(* CoDeSys 2.3.9.62 project: udptest.pro *)
(* Libraries: SysLibSocketsAsync.lib, SysLibSockets.lib, Standard.lib, Iecsfc.lib 8.11.10 11:37:48, SYSLIBCALLBACK.LIB *)

(* PLC configuration (modules and I/O channels)
K-Bus [K_Bus] node 0, in %IB0 out %QB0
Internal Digital I/O [InternalDigIO] node 1, in %IB512 out %QB512
  Internal Digital Inputs [Internal_DIN] node 0, in %IB512 out %QB512
    DIN1 AT %IX2300.0 [BOOLOnX_I] Internal Digital Input Bit 1
    DIN2 AT %IX2300.1 [BOOLOnX_I] Internal Digital Input Bit 2
  Internal Digital Outputs [Internal_DOUT] node 1, in %IB513 out %QB512
    DOUT1 AT %QX2300.0 [BOOLOnX_Q] Internal Digital Output Bit 1
    DOUT2 AT %QX2300.1 [BOOLOnX_Q] Internal Digital Output Bit 2
Fieldbus variables [FB_VARS] node 3, in %IB0 out %QB0
Flag variables [FLAG_VARS] node 4, in %IB0 out %QB0
Modbus-Master [MB_MASTER] node 5, in %IB0 out %QB0
*)

(* Task configuration *)
TASK RunMainProgram (PRIORITY := 15);
	PLC_PRG();
END_TASK

(* POU PLC_PRG, FBD *)
PROGRAM PLC_PRG
VAR
	Platform  : PLATFORM_SIMULATOR;
	Driver: MotorDriver;
	MotorAngles: ComputeMotorAngles;

	wanted_angle_1 : REAL;
	wanted_angle_2 : REAL;
	wanted_angle_3 : REAL;

	motor_counts_1 : DINT;
	motor_counts_2 : DINT;
	motor_counts_3 : DINT;

	limit_switch_1 : BOOL;
	limit_switch_2 : BOOL;
	limit_switch_3 : BOOL;

	roll : REAL;
	pitch : REAL;

	wanted_roll : REAL;
	wanted_pitch : REAL;
	UDPOK: FB_UDP_Receiver;

	test1 : BOOL;
	test2 : UDINT;
	test3 : DINT;

END_VAR
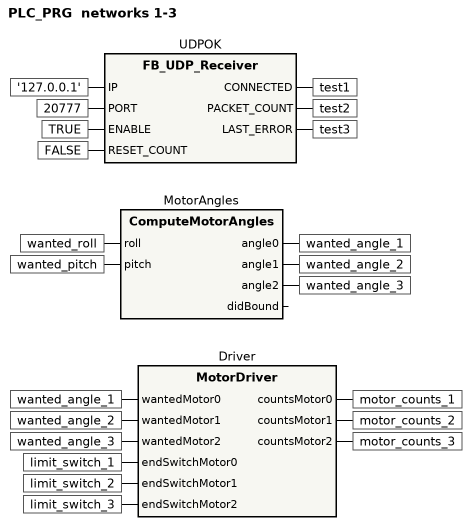
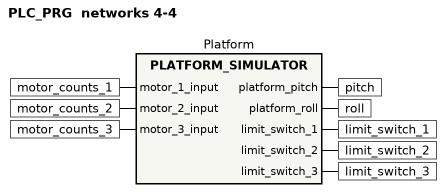
_FBD_ (* Function Block Diagram *)
NETWORK 1
	UDPOK:FB_UDP_Receiver(IP: '127.0.0.1', PORT: 20777, ENABLE: TRUE, RESET_COUNT: FALSE, PACKET_COUNT => test2, LAST_ERROR => test3) => test1
NETWORK 2
	MotorAngles:ComputeMotorAngles(roll: wanted_roll, pitch: wanted_pitch, angle1 => wanted_angle_2, angle2 => wanted_angle_3) => wanted_angle_1
NETWORK 3
	Driver:MotorDriver(wantedMotor0: wanted_angle_1, wantedMotor1: wanted_angle_2, wantedMotor2: wanted_angle_3, endSwitchMotor0: limit_switch_1, endSwitchMotor1: limit_switch_2, endSwitchMotor2: limit_switch_3, countsMotor1 => motor_counts_2, countsMotor2 => motor_counts_3) => motor_counts_1
NETWORK 4
	Platform:PLATFORM_SIMULATOR(motor_1_input: motor_counts_1, motor_2_input: motor_counts_2, motor_3_input: motor_counts_3, platform_roll => roll, limit_switch_1 => limit_switch_1, limit_switch_2 => limit_switch_2, limit_switch_3 => limit_switch_3) => pitch
_END_FBD_
(* the same logic as Structured Text *)
(* Network 1 *)
UDPOK(IP := '127.0.0.1', PORT := 20777, ENABLE := TRUE, RESET_COUNT := FALSE);
test2 := UDPOK.PACKET_COUNT;
test3 := UDPOK.LAST_ERROR;
test1 := UDPOK.CONNECTED;
(* Network 2 *)
MotorAngles(roll := wanted_roll, pitch := wanted_pitch);
wanted_angle_2 := MotorAngles.angle1;
wanted_angle_3 := MotorAngles.angle2;
wanted_angle_1 := MotorAngles.angle0;
(* Network 3 *)
Driver(wantedMotor0 := wanted_angle_1, wantedMotor1 := wanted_angle_2, wantedMotor2 := wanted_angle_3, endSwitchMotor0 := limit_switch_1, endSwitchMotor1 := limit_switch_2, endSwitchMotor2 := limit_switch_3);
motor_counts_2 := Driver.countsMotor1;
motor_counts_3 := Driver.countsMotor2;
motor_counts_1 := Driver.countsMotor0;
(* Network 4 *)
Platform(motor_1_input := motor_counts_1, motor_2_input := motor_counts_2, motor_3_input := motor_counts_3);
roll := Platform.platform_roll;
limit_switch_1 := Platform.limit_switch_1;
limit_switch_2 := Platform.limit_switch_2;
limit_switch_3 := Platform.limit_switch_3;
pitch := Platform.platform_pitch;
END_PROGRAM

(* POU PLATFORM_SIMULATOR, ST *)
FUNCTION_BLOCK PLATFORM_SIMULATOR
VAR_INPUT
	 motor_1_input  :  DINT;
   	 motor_2_input  :  DINT;
   	 motor_3_input  :  DINT;
END_VAR
VAR_OUTPUT
    	platform_pitch : REAL;
    	platform_roll : REAL;
	limit_switch_1 : BOOL;
	limit_switch_2 : BOOL;
	limit_switch_3 : BOOL;
END_VAR
VAR
	motor_1_angle : REAL;
	motor_2_angle : REAL;
    	motor_3_angle : REAL;
    	p1 : REAL;
    	p2 : REAL;
    	p3 : REAL;
END_VAR
motor_1_angle := motor_1_input * 0.0000392699;
motor_2_angle := motor_2_input * 0.0000392699;
motor_3_angle := motor_3_input * 0.0000392699;

limit_switch_1 := NOT((motor_1_angle > (350 * 0.01745328627) AND motor_1_angle < (359 * 0.01745328627)));
limit_switch_2 := NOT((motor_2_angle > (350 * 0.01745328627) AND motor_2_angle < (359 * 0.01745328627)));
limit_switch_3 := NOT((motor_3_angle > (350 * 0.01745328627) AND motor_3_angle < (359 * 0.01745328627)));

p1 := 0.08 * (1 - COS(motor_1_angle));
p2 := 0.08 * (1 - COS(motor_2_angle));
p3 := 0.08 * (1 - COS(motor_3_angle));

platform_pitch := ATAN((p2 - ((p3 + p1) / 2)) / ((1.75 * SQRT(3)) / 2));

platform_roll := ATAN((p3 - p1) / 1.75);
END_FUNCTION_BLOCK

(* POU MotorDriver, ST *)
FUNCTION_BLOCK MotorDriver
VAR_INPUT
	wantedMotor0: REAL;
	wantedMotor1: REAL;
	wantedMotor2: REAL;
	endSwitchMotor0: BOOL;
	endSwitchMotor1: BOOL;
	endSwitchMotor2: BOOL;
END_VAR
VAR_OUTPUT
	countsMotor0: DINT;
	countsMotor1: DINT;
	countsMotor2: DINT;
END_VAR
VAR
	endSwitchPosition: DINT := -10000;
END_VAR
IF endSwitchMotor0 THEN
	countsMotor0 := motorAngleToCounts(wantedMotor0);
ELSE
	countsMotor0 := 0;
END_IF
IF endSwitchMotor0 THEN
	countsMotor1 := motorAngleToCounts(wantedMotor1);
ELSE
	countsMotor1 := 0;
END_IF
IF endSwitchMotor0 THEN
	countsMotor2 := motorAngleToCounts(wantedMotor2);
ELSE
	countsMotor2 := 0;
END_IF
END_FUNCTION_BLOCK

(* POU motorAngleToCounts, ST *)
FUNCTION motorAngleToCounts : DINT
VAR_INPUT
	wantedMotorAngle: REAL;
END_VAR
VAR
	motorCountsPerRound: REAL := 160000;
	pi: REAL := 3.1415926;
	tempVar: DINT;
END_VAR
motorAngleToCounts := REAL_TO_DINT((wantedMotorAngle * motorCountsPerRound)/(2*pi));
END_FUNCTION

(* POU ComputeMotorAngles, ST *)
FUNCTION_BLOCK ComputeMotorAngles
VAR_INPUT
	roll : LREAL;
	pitch : LREAL;
END_VAR
VAR_OUTPUT
	angle0 : LREAL;
	angle1 : LREAL;
	angle2 : LREAL;

	didBound : BOOL;
END_VAR
VAR
	l : LREAL := 1.75;
	delta : LREAL := 0.08;
	s0 : LREAL := 1.0;
	s1 : LREAL := 1.0;

	tmpVar0 : LREAL;
	tmpVar1 : LREAL;

	p0 : LREAL;
	p1 : LREAL;
	p2 : LREAL;
END_VAR
tmpVar0 := l / 2 * ATAN(roll / s1);
p1 :=delta + tmpVar0;
p0 := delta - tmpVar0;

tmpVar1 := (l * SQRT(3) / 2) * ATAN(pitch / s0) / 2.0;
p2 := delta - tmpVar1;

p0 := p0 + tmpVar1;
p1 := p1 + tmpVar1;

p0 := -1.0 * (p0 - delta) / delta;
p1 := -1.0 * (p1 - delta) / delta;
p2 := -1.0 * (p2 - delta) / delta;

didBound := FALSE;

IF (p0 > 1.0) THEN
	p0 := 1.0;
	didBound := TRUE;
ELSIF (p0 < -1.0) THEN
	p0 := -1.0;
	didBound := TRUE;
END_IF


IF (p1 > 1.0) THEN
	p1 := 1.0;
	didBound := TRUE;
ELSIF (p1 < -1.0) THEN
	p1 := -1.0;
	didBound := TRUE;
END_IF

IF (p2 > 1.0) THEN
	p2 := 1.0;
	didBound := TRUE;
ELSIF (p2 < -1.0) THEN
	p2 := -1.0;
	didBound := TRUE;
END_IF

angle0 := ACOS(p0);
angle2 := ACOS(p1);
angle1 := ACOS(p2);
END_FUNCTION_BLOCK

(* POU FB_UDP_Receiver, ST *)
FUNCTION_BLOCK FB_UDP_Receiver
VAR_INPUT
    IP: STRING(15);
    PORT: UINT;
    ENABLE: BOOL;
    RESET_COUNT: BOOL;
END_VAR
VAR_OUTPUT
    CONNECTED: BOOL;
    PACKET_COUNT: UDINT;
    LAST_ERROR: DINT;
END_VAR
VAR
    hSocket: DINT := SOCKET_INVALID;
    localAddr: SOCKADDRESS;
    rxBuffer: ARRAY[0..1471] OF BYTE;
    bNonBlocking: BOOL := TRUE;
    dwIP: DWORD;
	fromAddr: SOCKADDRESS;
       fromLen: DINT;
       bytesReceived: DINT;
END_VAR
IF RESET_COUNT THEN
    PACKET_COUNT := 0;
END_IF

IF ENABLE THEN
    IF hSocket = SOCKET_INVALID THEN
        hSocket := SysSockCreate(
            diAddressFamily := SOCKET_AF_INET,
            diType := SOCKET_DGRAM,
            diProtocol := SOCKET_IPPROTO_UDP
        );

        IF hSocket <> SOCKET_INVALID THEN
            SysSockIoctl(
                diSocket := hSocket,
                diCommand := SOCKET_FIONBIO,
                piParameter := ADR(bNonBlocking)
            );

            dwIP := SysSockInetAddr(IP);
            IF IP = '0.0.0.0' THEN
                dwIP := SOCKET_INADDR_ANY;
            END_IF;

            localAddr.sin_family := SOCKET_AF_INET;
            localAddr.sin_port := SysSockHtons(PORT);
            localAddr.sin_addr := dwIP;

            IF NOT SysSockBind(diSocket := hSocket, pSockAddr := ADR(localAddr), diSockAddrSize := SIZEOF(localAddr)) THEN
                LAST_ERROR := SysSockGetLastErrorSync(hSocket);
                SysSockClose(hSocket);
                hSocket := SOCKET_INVALID;
            END_IF;
        END_IF;
    END_IF;

    CONNECTED := (hSocket <> SOCKET_INVALID);

    fromLen:= SIZEOF(fromAddr);

    IF CONNECTED THEN

        bytesReceived := SysSockRecvFrom(
            diSocket := hSocket,
            pbyBuffer := ADR(rxBuffer),
            diBufferSize := SIZEOF(rxBuffer),
            diFlags := 0,
            pSockAddr := ADR(fromAddr),
            diSockAddrSize := fromLen
        );
        
        IF bytesReceived > 0 THEN
            PACKET_COUNT := PACKET_COUNT + 1;
        ELSIF bytesReceived < 0 THEN
            LAST_ERROR := SysSockGetLastErrorSync(hSocket);
        END_IF;
    END_IF;
ELSE
    IF hSocket <> SOCKET_INVALID THEN
        SysSockClose(hSocket);
        hSocket := SOCKET_INVALID;
    END_IF;
    CONNECTED := FALSE;
END_IF;
END_FUNCTION_BLOCK

(* POU UDPDecoder, ST *)
FUNCTION_BLOCK UDPDecoder
VAR_INPUT
	initialData: STRING(528);
END_VAR
VAR_OUTPUT
	floatArray : ARRAY [0..66] OF REAL;
END_VAR
VAR
   	hexSeperated: ARRAY[0..66] OF STRING(8);
	reversedHexSeperated: ARRAY[0..66] OF STRING(8);
	hexAsInt: ARRAY[0..66] OF REAL		(*Må være real for at EXPT funksjonen skal funke*);
	numberToMakeBinary: DWORD;
	binaryHexAsInt: ARRAY[0..66] OF ARRAY[0..31] OF BOOL;
 	i: INT;
	j: INT;
	k: INT;
	iterationCounter: INT := 0;
	calculationInt: INT;
	sign: INT;
	exponent: REAL;
	mantissa: REAL;
	hexArray: ARRAY[0..15] OF STRING(1);

END_VAR
(*Konvertering av little endian hexadecimal til flyttall*)
(*Usexy kode, finn ut hvordan det kan deklareres i deklareringsområdet*)
IF iterationCounter = 0 THEN
	hexArray[0] := '0';
	hexArray[1] := '1';
	hexArray[2] := '2';
	hexArray[3] := '3';
	hexArray[4] := '4';
	hexArray[5] := '5';
	hexArray[6] := '6';
	hexArray[7] := '7';
	hexArray[8] := '8';
	hexArray[9] := '9';
	hexArray[10] := 'a';
	hexArray[11] := 'b';
	hexArray[12] := 'c';
	hexArray[13] := 'd';
	hexArray[14] := 'e';
	hexArray[15] := 'f';

	(*Deler den oprinnlige tekststrengen opp i de forskjellige verdiene*)
	FOR i := 0 TO 66 DO
	    hexSeperated[i] := MID(initialData, 8, (i * 8) + 1);
	END_FOR

	(*Snur strengene for å passe med little endian*)
	FOR i := 0 TO 66 DO
		FOR j := 0 TO 7 BY 2 DO
			reversedHexSeperated[i] := CONCAT( reversedHexSeperated[i],  MID(hexSeperated[i], 2, 8 - j - 1));
		END_FOR
	END_FOR

	(*Regner ut  desimalen som hører til hexadesimalen*)
	FOR i := 0 TO 66 DO
		hexAsInt[i] := 0;
		FOR j := 0 TO 7 DO
			FOR k := 0 TO 15 DO
				IF MID(reversedHexSeperated[i], 1, j + 1) = hexArray[k] THEN
					hexAsInt[i] := hexAsInt[i] + k * EXPT(16, 7 - j);
					EXIT;
				END_IF
			END_FOR
		END_FOR
	END_FOR

	(*Gjør inten om til binært for å kunne regne ut mantissa, eksponent og sign*)
	FOR i := 0 TO 66 DO
		numberToMakeBinary := REAL_TO_DWORD(hexAsInt[i]);
		FOR j := 0 TO 31 DO
			binaryHexAsInt[i][j] := (numberToMakeBinary AND 16#80000000) <> 0;
			numberToMakeBinary := SHL(numberToMakeBinary, 1);
		END_FOR
	END_FOR

	(*Regner ut sign, eksponent og mantissa*)
	FOR i := 0 TO 66 DO
		sign := 0;
		exponent := 0;
		mantissa := 0;
		(*Sjekker første binærtallet for å finne ut om det er positivt eller negativt*)
		IF NOT binaryHexAsInt[i][0] THEN
			sign := 0;
		ELSE
			sign := 1;
		END_IF
		(*Regner ut eksponenten for fra binærtallet*)
		FOR j := 1 TO 8 DO
            		IF binaryHexAsInt[i][j] THEN
                		exponent := exponent + EXPT(2, 8 - j);
	            END_IF
        	END_FOR
        	exponent := exponent - 127;
		(*Regner ut mantissaen med de resterende talla i binærtallet*)
		FOR j := 9 TO 31 DO
            		IF binaryHexAsInt[i][j] THEN
                		mantissa := mantissa + EXPT(2, 8 - j);
	            END_IF
       	 END_FOR

		floatArray[i] := EXPT(-1, sign) * (1.0 + mantissa) * EXPT(2, exponent);
	END_FOR

	iterationCounter := iterationCounter + 1;
END_IF
END_FUNCTION_BLOCK
